// TIA Portal V17 export
// export: Created 2026-07-06T15:33:04.9330509Z, ExportSetting WithDefaults, DisplayName Totally Integrated Automation Portal, DisplayVersion V17, DisplayName TIA Portal Openness, DisplayVersion V17, DisplayName TIA Portal Version Control Interface, DisplayVersion V17, DisplayName STEP 7 Professional, DisplayVersion V17, DisplayName STEP 7 Safety, DisplayVersion V17, DisplayName WinCC Professional, DisplayVersion V17
DATA_BLOCK "PULSE_TIMER_DB_move_pulse"   // DB2
VERSION : 0.1
// stored: AutoNumber true, DBAccessibleFromOPCUA true, InstanceOfName PULSE_TIMER, InstanceOfType FB
"PULSE_TIMER"
   // VAR_INPUT
   //    "PULSE HZ" : Real;
   // END_VAR
   // VAR_OUTPUT
   //    PULSE : Bool;
   // END_VAR
   // VAR
   //    Clock_Timer_1 : IEC_TIMER;
   //    Clock_Timer_2 : IEC_TIMER;
   //    "Time(s)" { S7_SetPoint := 'True'} : Real;
   //    "Time(ms)" : Real;
   //    "Time" : Int;
   // END_VAR
BEGIN
END_DATA_BLOCK
